(* Logix 5000 project; controller DispersionPlc vendor 1 type 14 code 108 rev 34.11; software revision 34.01; part 5 of 22 *)
(* tags used below, declared in another part *)
   catalyst_Target_Wgt_Lb_Min : REAL;
   D_Alarm_11_Timer : TIMER;
   D_Alarm_9_Timer : TIMER;
   D_AlarmTimers : TIMER[200];
   D_AlarmTimers2 : TIMER[100];
   DPT_4303_Warn : REAL;
   ONS : BOOL[32];
   ZS_4301_timer : TIMER;
   ZS_4302_timer : TIMER;
   _JISdebug : DINT;
   AFB : BOOL;
   AFI : BOOL;
   AMMONIUM_START_ATTEMP : BOOL;
   BL_4310_AUX : ALIAS FOR Local:1:I.Data[1].2;
   BL_4310_RUN : ALIAS FOR Local:1:O.Data[0].2;
   BLANK64 : Stp64;
   Cat_Destination_K400 : BOOL;
   Cat_Destination_K400_ONS : BOOL;
   Cat_Destination_K400_PB : BOOL;
   Cat_Destination_T4301 : BOOL;
   Cat_Destination_T4301_ONS : BOOL;
   Cat_Destination_T4301_PB : BOOL;
   Cat_Isolation_Valve_Timer : TIMER;
   Cat_Purge_Transfer_K400 : Seq64;
   Cat_Purge_Transfer_T430X : Seq64;
   Cat_Recirc_Transfer_K400 : Seq64;
   Cat_Recirc_Transfer_T430X : Seq64;
   Cat_Tank_Destination : DINT;
   cat_target_weight_bypass : BOOL;
   catalyst_MaxFeedRate : REAL;
   CATALYST_RESET : BOOL;
   CATFLOW : TIMER;
   CE_4301 : REAL;
   ce_4301_High : REAL;
   ce_4301_Low : REAL;
   DispAlarmResetBit : BOOL;
   DispersionAlarms : BOOL[256];
   DPT_4301 : REAL;
   dpt_4301_High : REAL;
   DPT_4302 : REAL;
   dpt_4302_High : REAL;
   DPT_4303 : REAL;
   DPT_4303_High : REAL;
   Drum_Transfer : BOOL;
   Enable_Shortstop_Automation : BOOL;
   Estop_Bulk : ALIAS FOR Local:1:I.Data[33].5;
   Estop_Disp : ALIAS FOR Local:3:I.Data.1;
   Estop_Inx : ALIAS FOR Local:3:I.Data.3;
   Estop_Mcc : ALIAS FOR Local:3:I.Data.2;
   FE_4303 : REAL;
   FE_4303_Low : REAL;
   FE_4304 : REAL;
   FE_4304_Low : REAL;
   FE_4305 : REAL;
   FE_4305_LOW : REAL;
   GLOBAL_RESET : BOOL;
   HMI_4303_Timer : REAL;
   HMI_4304_Timer : REAL;
   HMI_Cat_Isolation_Valve_Timer : REAL;
   HMI_V4304_PumpSpeedScaleIn : REAL;
   K4_High_Temp : BOOL;
   K4_Low_Temp : BOOL;
   LAH_S4352_1 : ALIAS FOR Local:1:I.Data[27].13;
   Linked_Timer : TIMER;
   LS_4301 : ALIAS FOR Local:2:I.Data.10;
   LS_4302 : ALIAS FOR Local:2:I.Data.11;
   LS_4302_High : BOOL;
   LS_T53_High : ALIAS FOR Local:1:I.Data[27].12;
   MCR_Bulk : ALIAS FOR Local:1:I.Data[33].4;
   MIXER_A_4301_RUN : ALIAS FOR Local:1:O.Data[0].0;
   MIXER_A_4303_AUX : ALIAS FOR Local:1:I.Data[1].4;
   MIXER_A_4303_RUN : ALIAS FOR Local:1:O.Data[0].4;
   MIXER_A_4304_AUX : ALIAS FOR Local:1:I.Data[1].16;
   MIXER_A_4304_RUN : ALIAS FOR Local:1:O.Data[0].16;
   MIXER_T_4301_AUX : ALIAS FOR Local:1:I.Data[1].0;
   MMI_Disp_Alarm_Reset_Pb : BOOL;
   MMI_Dispersion_Interlock_Bypass : BOOL;
   Mon_Tank_Destination : DINT;
   PS_AirMakeup : ALIAS FOR Local:1:I.Data[33].3;
   PUMP_P_4305_AUX : ALIAS FOR Local:1:I.Data[1].7;
   PUMP_P_4305_RUN : ALIAS FOR Local:1:O.Data[0].7;
   RG_T52 : REAL;
   RG_T52_Warn : REAL;
   RG_T53 : REAL;
   RG_T53_Warn : REAL;
   SPARE_I304 : ALIAS FOR Local:3:I.Data.4;
   SPARE_I305 : ALIAS FOR Local:3:I.Data.5;
   SPARE_O510 : ALIAS FOR Local:5:O.Data.10;
   SRT_PB_BL_4310 : ALIAS FOR Local:2:I.Data.13;
   ST_K400_1 : REAL;
   SV_4304 : ALIAS FOR Local:5:O.Data.11;
   SV_4304_02 : BOOL;
   SV_4304_02_Enable_PB : BOOL;
   SV_4304_03 : BOOL;
   SV_4304_03_Enable_PB : BOOL;
   T4301_Mixer : VFD;
   T4302_Mixer : VFD;
   T52_Mixer : VFD;
   Tank_Destination_ONS1 : BOOL;
   Task_Permissive : DINT[2];
   TE_4301A : ALIAS FOR Local:8:I.Ch0Data;
   Te_4301A_High : REAL;
   TE_4302A : ALIAS FOR Local:8:I.Ch5Data;
   TE_4302A_High : REAL;
   TE_4304 : ALIAS FOR Local:9:I.Ch5Data;
   TE_4304_High : REAL;
   TO_ALARM_MSG_DINT : DINT;
   TOGGLE : BOOL;
   Trans_Pump_P52_Aux : ALIAS FOR Local:1:I.Data[33].0;
   Trans_Pump_P53_Aux : ALIAS FOR Local:1:I.Data[33].1;
   TRANS_PUMP_P_4301_AUX : ALIAS FOR Local:1:I.Data[1].1;
   TRANS_PUMP_P_4301_RUN : ALIAS FOR Local:1:O.Data[0].1;
   TRANS_PUMP_P_4302_AUX : ALIAS FOR Local:1:I.Data[1].3;
   TRANS_PUMP_P_4302_RUN : ALIAS FOR Local:1:O.Data[0].3;
   Trans_Pump_T52_Run : ALIAS FOR Local:1:O.Data[13].1;
   Trans_Pump_T53_Run : ALIAS FOR Local:1:O.Data[13].2;
   V4304_Pump : VFD;
   W4303_Pump : VFD;
   XI_K400_1 : BOOL;
   XV_4301 : ALIAS FOR Local:5:O.Data.0;
   XV_4302 : ALIAS FOR Local:5:O.Data.1;
   XV_4303_01 : ALIAS FOR Local:5:O.Data.3;
   XV_4304 : ALIAS FOR Local:5:O.Data.4;
   XV_4304_02 : BOOL;
   XV_4304_03 : BOOL;
   XV_4304_04 : BOOL;
   XV_5201 : ALIAS FOR Local:1:O.Data[12].8;
   XV_5202 : ALIAS FOR Local:1:O.Data[12].9;
   XV_5301 : ALIAS FOR Local:1:O.Data[12].6;
   XV_5302 : ALIAS FOR Local:1:O.Data[12].7;
   XV_K400_04_SEQCLOSE : BOOL;
   XV_K400_04_SEQOPEN : BOOL;
   ZSC_4301 : ALIAS FOR Local:2:I.Data.1;
   ZSC_4302 : ALIAS FOR Local:2:I.Data.3;
   ZSC_4303_1 : ALIAS FOR Local:2:I.Data.7;
   ZSC_4304 : ALIAS FOR Local:2:I.Data.9;
   ZSC_4304_02 : BOOL;
   ZSC_4304_03 : BOOL;
   ZSC_5201 : ALIAS FOR Local:1:I.Data[27].5;
   ZSC_5202 : ALIAS FOR Local:1:I.Data[27].7;
   ZSC_5301 : ALIAS FOR Local:1:I.Data[27].9;
   ZSC_5302 : ALIAS FOR Local:1:I.Data[27].11;
   ZSC_K400_04 : BOOL;
   ZSO_4301 : ALIAS FOR Local:2:I.Data.0;
   ZSO_4302 : ALIAS FOR Local:2:I.Data.2;
   ZSO_4303_1 : ALIAS FOR Local:2:I.Data.6;
   ZSO_4304 : ALIAS FOR Local:2:I.Data.8;
   ZSO_4304_02 : BOOL;
   ZSO_4304_03 : BOOL;
   ZSO_4304_04 : BOOL;
   ZSO_5201 : ALIAS FOR Local:1:I.Data[27].4;
   ZSO_5202 : ALIAS FOR Local:1:I.Data[27].6;
   ZSO_5301 : ALIAS FOR Local:1:I.Data[27].8;
   ZSO_5302 : ALIAS FOR Local:1:I.Data[27].10;
   ZSO_K400_04 : BOOL;
(* MainProgram, continued *)

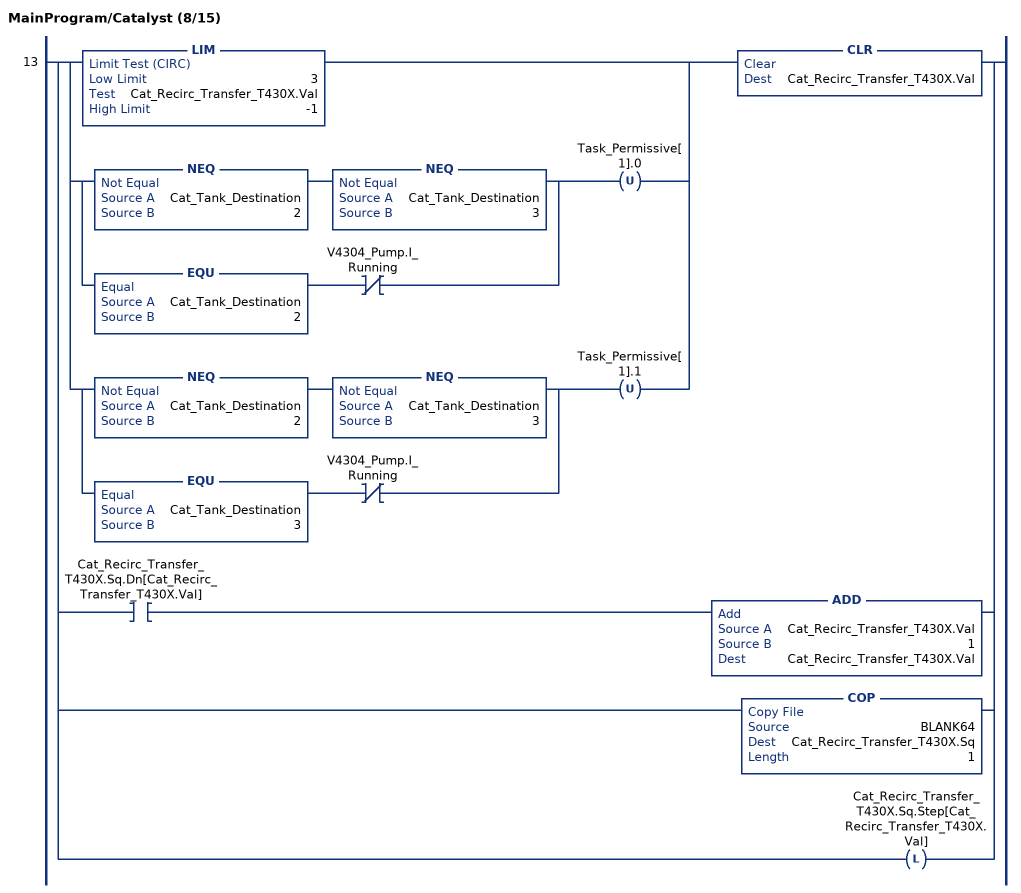
   [picture p69: MainProgram/Catalyst rungs 13-13]
   13: [[LIM(3,Cat_Recirc_Transfer_T430X.Val,-1) ,[NEQ(Cat_Tank_Destination,2) NEQ(Cat_Tank_Destination,3) ,EQU(Cat_Tank_Destination,2) XIO(V4304_Pump.I_Running) ] OTU(Task_Permissive[1].0) ,[NEQ(Cat_Tank_Destination,2) NEQ(Cat_Tank_Destination,3) ,EQU(Cat_Tank_Destination,3) XIO(V4304_Pump.I_Running) ] OTU(Task_Permissive[1].1) ] CLR(Cat_Recirc_Transfer_T430X.Val) ,XIC(Cat_Recirc_Transfer_T430X.Sq.Dn[Cat_Recirc_Transfer_T430X.Val]) ADD(Cat_Recirc_Transfer_T430X.Val,1,Cat_Recirc_Transfer_T430X.Val) ,COP(BLANK64,Cat_Recirc_Transfer_T430X.Sq,1) ,OTL(Cat_Recirc_Transfer_T430X.Sq.Step[Cat_Recirc_Transfer_T430X.Val]) ];
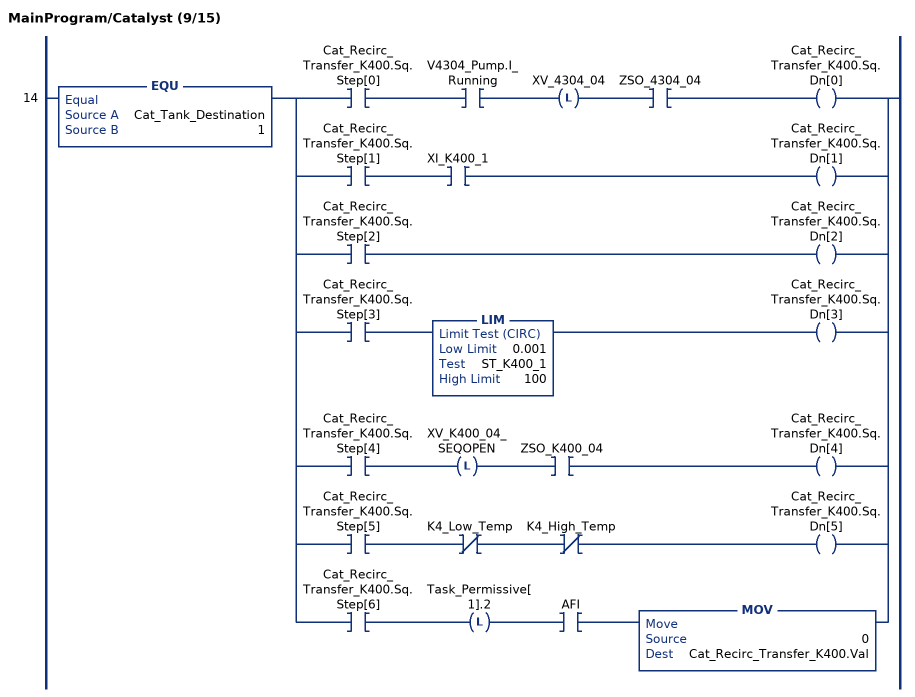
   14: EQU(Cat_Tank_Destination,1)[XIC(Cat_Recirc_Transfer_K400.Sq.Step[0]) XIC(V4304_Pump.I_Running) OTL(XV_4304_04) XIC(ZSO_4304_04) OTE(Cat_Recirc_Transfer_K400.Sq.Dn[0]) ,XIC(Cat_Recirc_Transfer_K400.Sq.Step[1]) XIC(XI_K400_1) OTE(Cat_Recirc_Transfer_K400.Sq.Dn[1]) ,XIC(Cat_Recirc_Transfer_K400.Sq.Step[2]) OTE(Cat_Recirc_Transfer_K400.Sq.Dn[2]) ,XIC(Cat_Recirc_Transfer_K400.Sq.Step[3]) LIM(0.001,ST_K400_1,100) OTE(Cat_Recirc_Transfer_K400.Sq.Dn[3]) ,XIC(Cat_Recirc_Transfer_K400.Sq.Step[4]) OTL(XV_K400_04_SEQOPEN) XIC(ZSO_K400_04) OTE(Cat_Recirc_Transfer_K400.Sq.Dn[4]) ,XIC(Cat_Recirc_Transfer_K400.Sq.Step[5]) XIO(K4_Low_Temp) XIO(K4_High_Temp) OTE(Cat_Recirc_Transfer_K400.Sq.Dn[5]) ,XIC(Cat_Recirc_Transfer_K400.Sq.Step[6]) OTL(Task_Permissive[1].2) XIC(AFI) MOV(0,Cat_Recirc_Transfer_K400.Val) ];
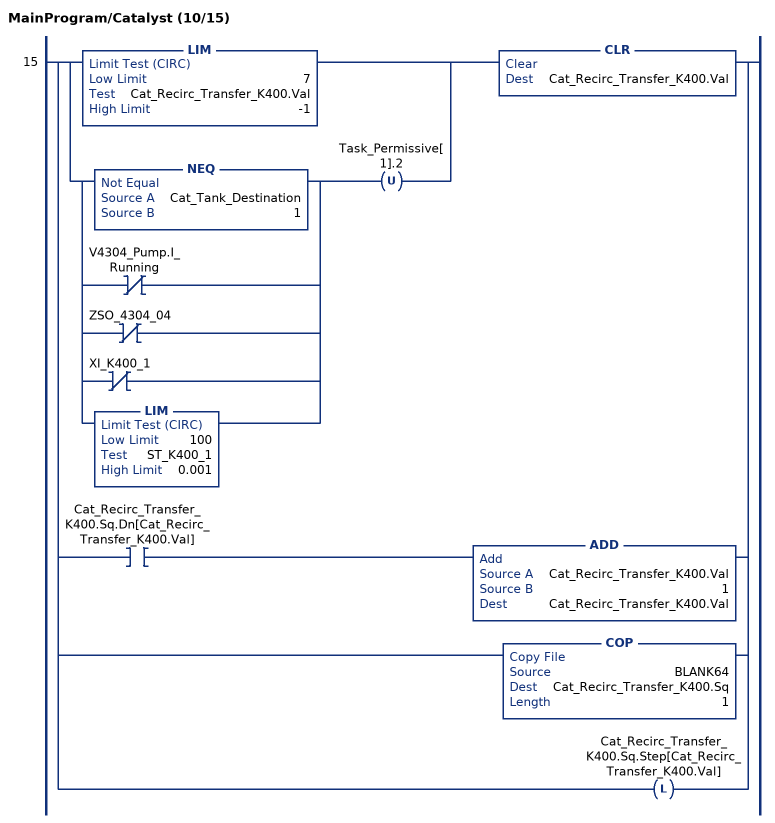
   15: [[LIM(7,Cat_Recirc_Transfer_K400.Val,-1) ,[NEQ(Cat_Tank_Destination,1) ,XIO(V4304_Pump.I_Running) ,XIO(ZSO_4304_04) ,XIO(XI_K400_1) ,LIM(100,ST_K400_1,0.001) ] OTU(Task_Permissive[1].2) ] CLR(Cat_Recirc_Transfer_K400.Val) ,XIC(Cat_Recirc_Transfer_K400.Sq.Dn[Cat_Recirc_Transfer_K400.Val]) ADD(Cat_Recirc_Transfer_K400.Val,1,Cat_Recirc_Transfer_K400.Val) ,COP(BLANK64,Cat_Recirc_Transfer_K400.Sq,1) ,OTL(Cat_Recirc_Transfer_K400.Sq.Step[Cat_Recirc_Transfer_K400.Val]) ];
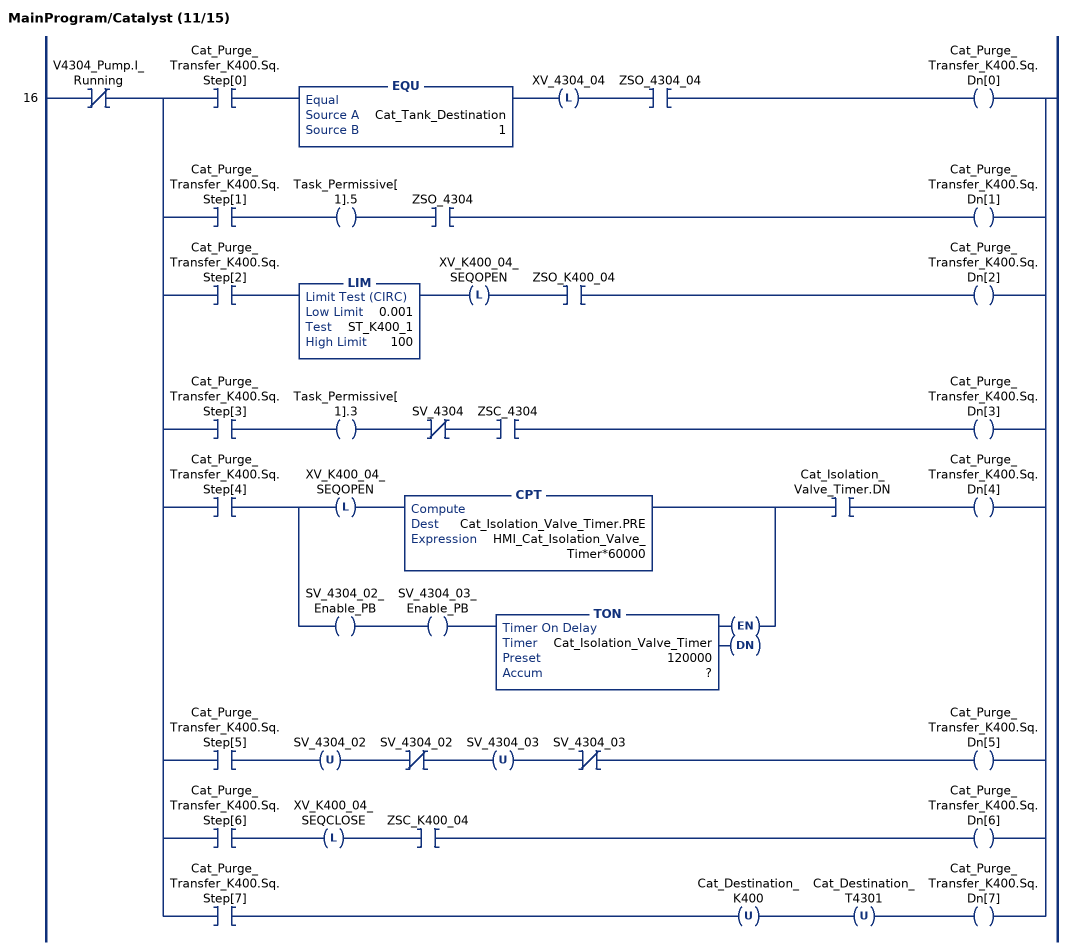
   16: XIO(V4304_Pump.I_Running)[XIC(Cat_Purge_Transfer_K400.Sq.Step[0]) EQU(Cat_Tank_Destination,1) OTL(XV_4304_04) XIC(ZSO_4304_04) OTE(Cat_Purge_Transfer_K400.Sq.Dn[0]) ,XIC(Cat_Purge_Transfer_K400.Sq.Step[1]) OTE(Task_Permissive[1].5) XIC(ZSO_4304) OTE(Cat_Purge_Transfer_K400.Sq.Dn[1]) ,XIC(Cat_Purge_Transfer_K400.Sq.Step[2]) LIM(0.001,ST_K400_1,100) OTL(XV_K400_04_SEQOPEN) XIC(ZSO_K400_04) OTE(Cat_Purge_Transfer_K400.Sq.Dn[2]) ,XIC(Cat_Purge_Transfer_K400.Sq.Step[3]) OTE(Task_Permissive[1].3) XIO(SV_4304) XIC(ZSC_4304) OTE(Cat_Purge_Transfer_K400.Sq.Dn[3]) ,XIC(Cat_Purge_Transfer_K400.Sq.Step[4]) [OTL(XV_K400_04_SEQOPEN) CPT(Cat_Isolation_Valve_Timer.PRE,HMI_Cat_Isolation_Valve_Timer*60000) ,OTE(SV_4304_02_Enable_PB) OTE(SV_4304_03_Enable_PB) TON(Cat_Isolation_Valve_Timer,?,?) ] XIC(Cat_Isolation_Valve_Timer.DN) OTE(Cat_Purge_Transfer_K400.Sq.Dn[4]) ,XIC(Cat_Purge_Transfer_K400.Sq.Step[5]) OTU(SV_4304_02) XIO(SV_4304_02) OTU(SV_4304_03) XIO(SV_4304_03) OTE(Cat_Purge_Transfer_K400.Sq.Dn[5]) ,XIC(Cat_Purge_Transfer_K400.Sq.Step[6]) OTL(XV_K400_04_SEQCLOSE) XIC(ZSC_K400_04) OTE(Cat_Purge_Transfer_K400.Sq.Dn[6]) ,XIC(Cat_Purge_Transfer_K400.Sq.Step[7]) OTU(Cat_Destination_K400) OTU(Cat_Destination_T4301) OTE(Cat_Purge_Transfer_K400.Sq.Dn[7]) ];
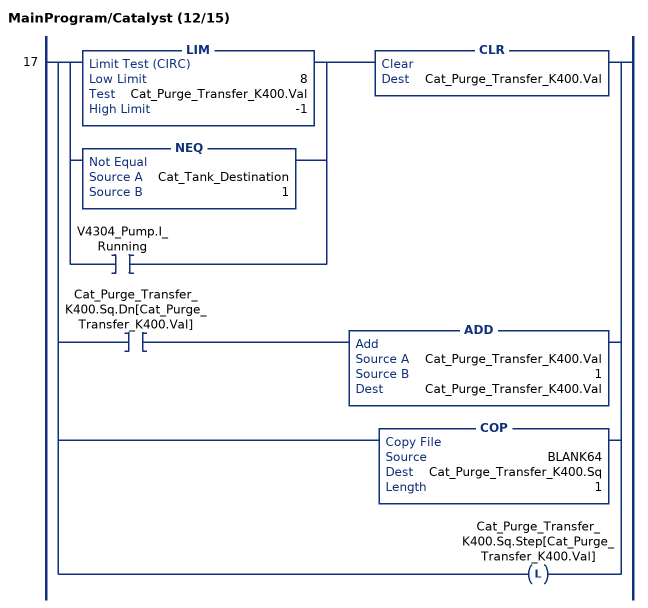
   17: [[LIM(8,Cat_Purge_Transfer_K400.Val,-1) ,NEQ(Cat_Tank_Destination,1) ,XIC(V4304_Pump.I_Running) ] CLR(Cat_Purge_Transfer_K400.Val) ,XIC(Cat_Purge_Transfer_K400.Sq.Dn[Cat_Purge_Transfer_K400.Val]) ADD(Cat_Purge_Transfer_K400.Val,1,Cat_Purge_Transfer_K400.Val) ,COP(BLANK64,Cat_Purge_Transfer_K400.Sq,1) ,OTL(Cat_Purge_Transfer_K400.Sq.Step[Cat_Purge_Transfer_K400.Val]) ];
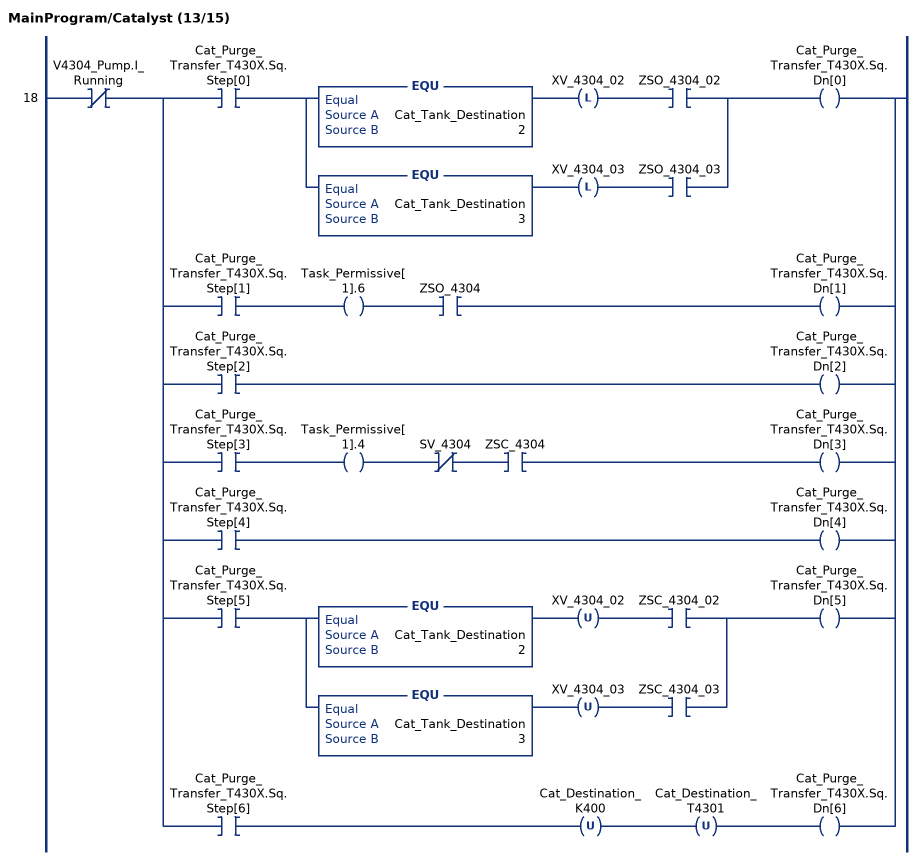
   18: XIO(V4304_Pump.I_Running)[XIC(Cat_Purge_Transfer_T430X.Sq.Step[0]) [EQU(Cat_Tank_Destination,2) OTL(XV_4304_02) XIC(ZSO_4304_02) ,EQU(Cat_Tank_Destination,3) OTL(XV_4304_03) XIC(ZSO_4304_03) ] OTE(Cat_Purge_Transfer_T430X.Sq.Dn[0]) ,XIC(Cat_Purge_Transfer_T430X.Sq.Step[1]) OTE(Task_Permissive[1].6) XIC(ZSO_4304) OTE(Cat_Purge_Transfer_T430X.Sq.Dn[1]) ,XIC(Cat_Purge_Transfer_T430X.Sq.Step[2]) OTE(Cat_Purge_Transfer_T430X.Sq.Dn[2]) ,XIC(Cat_Purge_Transfer_T430X.Sq.Step[3]) OTE(Task_Permissive[1].4) XIO(SV_4304) XIC(ZSC_4304) OTE(Cat_Purge_Transfer_T430X.Sq.Dn[3]) ,XIC(Cat_Purge_Transfer_T430X.Sq.Step[4]) OTE(Cat_Purge_Transfer_T430X.Sq.Dn[4]) ,XIC(Cat_Purge_Transfer_T430X.Sq.Step[5]) [EQU(Cat_Tank_Destination,2) OTU(XV_4304_02) XIC(ZSC_4304_02) ,EQU(Cat_Tank_Destination,3) OTU(XV_4304_03) XIC(ZSC_4304_03) ] OTE(Cat_Purge_Transfer_T430X.Sq.Dn[5]) ,XIC(Cat_Purge_Transfer_T430X.Sq.Step[6]) OTU(Cat_Destination_K400) OTU(Cat_Destination_T4301) OTE(Cat_Purge_Transfer_T430X.Sq.Dn[6]) ];
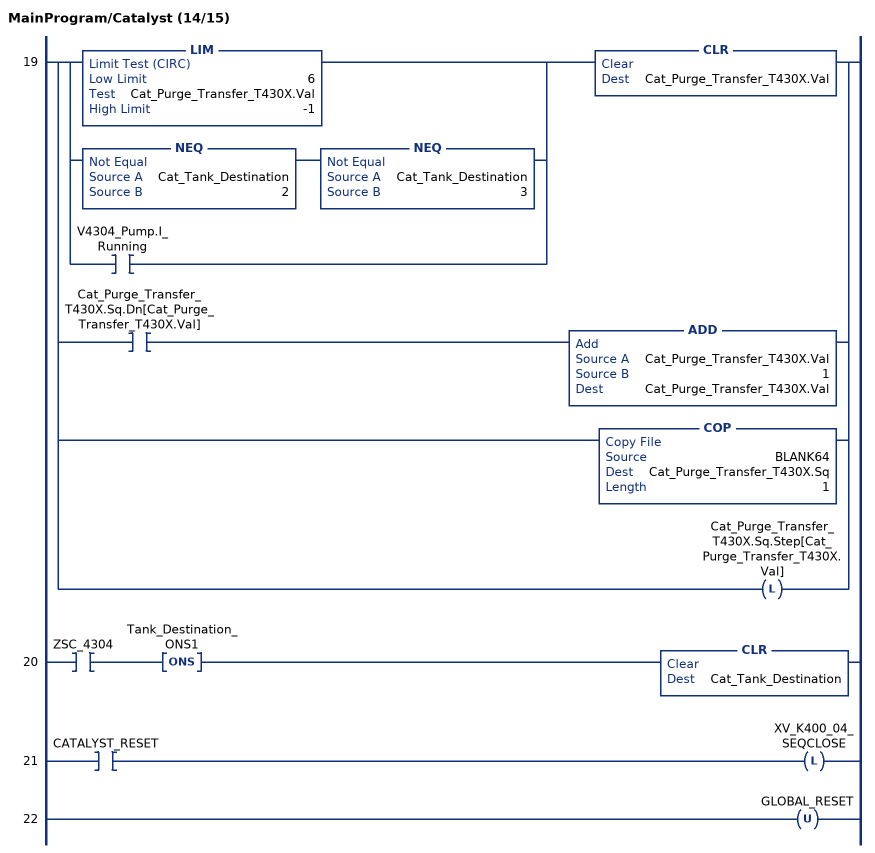
   19: [[LIM(6,Cat_Purge_Transfer_T430X.Val,-1) ,NEQ(Cat_Tank_Destination,2) NEQ(Cat_Tank_Destination,3) ,XIC(V4304_Pump.I_Running) ] CLR(Cat_Purge_Transfer_T430X.Val) ,XIC(Cat_Purge_Transfer_T430X.Sq.Dn[Cat_Purge_Transfer_T430X.Val]) ADD(Cat_Purge_Transfer_T430X.Val,1,Cat_Purge_Transfer_T430X.Val) ,COP(BLANK64,Cat_Purge_Transfer_T430X.Sq,1) ,OTL(Cat_Purge_Transfer_T430X.Sq.Step[Cat_Purge_Transfer_T430X.Val]) ];
   20: XIC(ZSC_4304)ONS(Tank_Destination_ONS1)CLR(Cat_Tank_Destination);
   21: XIC(CATALYST_RESET)OTL(XV_K400_04_SEQCLOSE);
   22: OTU(GLOBAL_RESET);
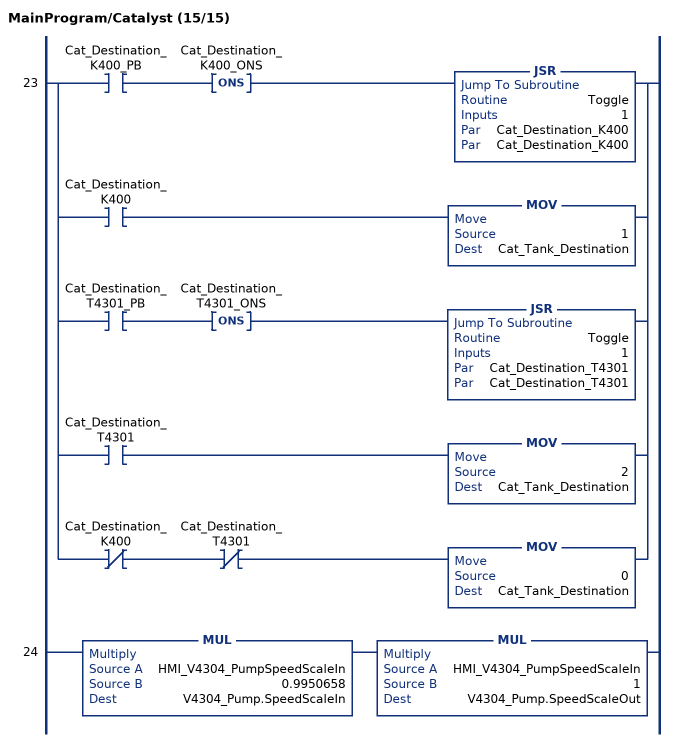
   23: [[XIC(Cat_Destination_K400_PB) ONS(Cat_Destination_K400_ONS) JSR(Toggle,1,Cat_Destination_K400,Cat_Destination_K400) ,XIC(Cat_Destination_K400) MOV(1,Cat_Tank_Destination) ] ,[XIC(Cat_Destination_T4301_PB) ONS(Cat_Destination_T4301_ONS) JSR(Toggle,1,Cat_Destination_T4301,Cat_Destination_T4301) ,XIC(Cat_Destination_T4301) MOV(2,Cat_Tank_Destination) ] ,XIO(Cat_Destination_K400) XIO(Cat_Destination_T4301) MOV(0,Cat_Tank_Destination) ];
   24: MUL(HMI_V4304_PumpSpeedScaleIn,0.9950658,V4304_Pump.SpeedScaleIn)MUL(HMI_V4304_PumpSpeedScaleIn,1,V4304_Pump.SpeedScaleOut);
END_ROUTINE

ROUTINE Dispersion_Alarms   (* ladder *)
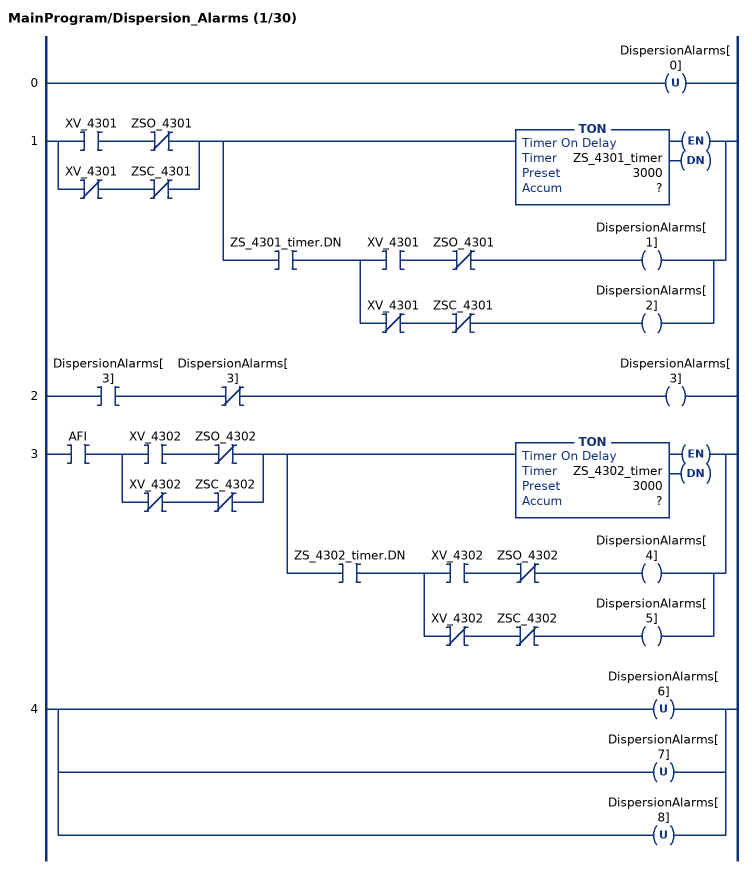
   0: OTU(DispersionAlarms[0]);
   1: [XIC(XV_4301) XIO(ZSO_4301) ,XIO(XV_4301) XIO(ZSC_4301) ][TON(ZS_4301_timer,?,?) ,XIC(ZS_4301_timer.DN) [XIC(XV_4301) XIO(ZSO_4301) OTE(DispersionAlarms[1]) ,XIO(XV_4301) XIO(ZSC_4301) OTE(DispersionAlarms[2]) ] ];
   2: XIC(DispersionAlarms[3])XIO(DispersionAlarms[3])OTE(DispersionAlarms[3]);
   3: XIC(AFI)[XIC(XV_4302) XIO(ZSO_4302) ,XIO(XV_4302) XIO(ZSC_4302) ][TON(ZS_4302_timer,?,?) ,XIC(ZS_4302_timer.DN) [XIC(XV_4302) XIO(ZSO_4302) OTE(DispersionAlarms[4]) ,XIO(XV_4302) XIO(ZSC_4302) OTE(DispersionAlarms[5]) ] ];
   4: [OTU(DispersionAlarms[6]) ,OTU(DispersionAlarms[7]) ,OTU(DispersionAlarms[8]) ];
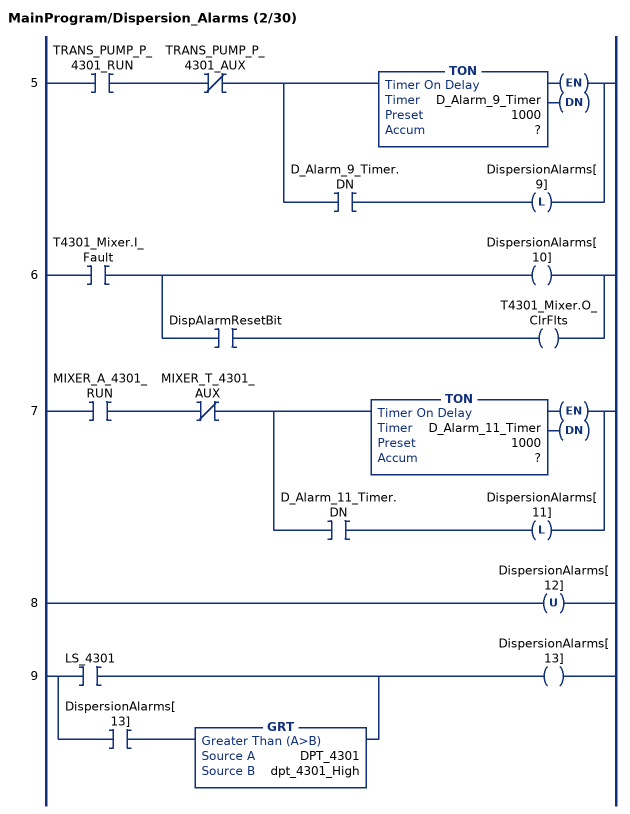
   5: XIC(TRANS_PUMP_P_4301_RUN)XIO(TRANS_PUMP_P_4301_AUX)[TON(D_Alarm_9_Timer,?,?) ,XIC(D_Alarm_9_Timer.DN) OTL(DispersionAlarms[9]) ];
   6: XIC(T4301_Mixer.I_Fault)[OTE(DispersionAlarms[10]) ,XIC(DispAlarmResetBit) OTE(T4301_Mixer.O_ClrFlts) ];
   7: XIC(MIXER_A_4301_RUN)XIO(MIXER_T_4301_AUX)[TON(D_Alarm_11_Timer,?,?) ,XIC(D_Alarm_11_Timer.DN) OTL(DispersionAlarms[11]) ];
   8: OTU(DispersionAlarms[12]);
   9: [XIC(LS_4301) ,XIC(DispersionAlarms[13]) GRT(DPT_4301,dpt_4301_High) ]OTE(DispersionAlarms[13]);
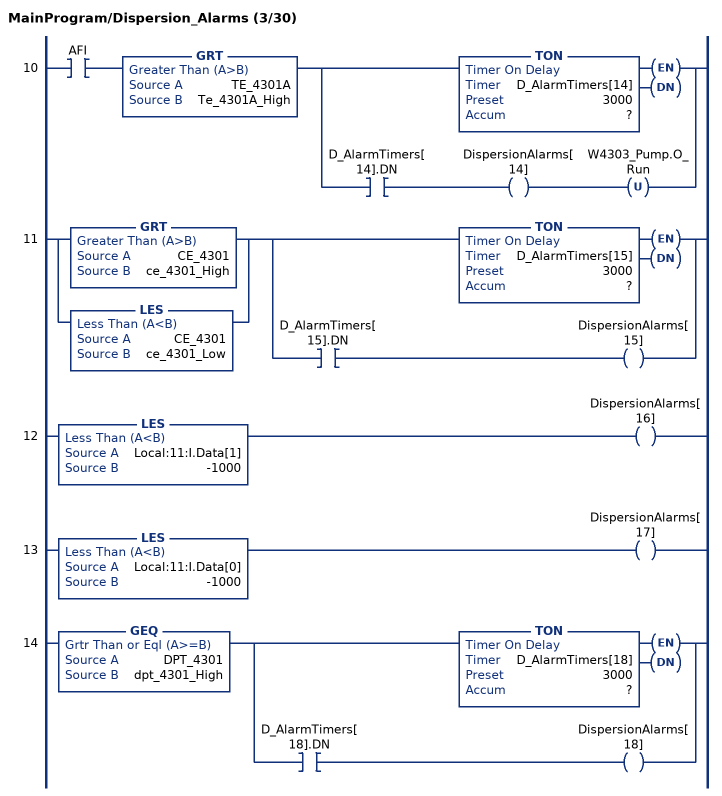
   10: XIC(AFI)GRT(TE_4301A,Te_4301A_High)[TON(D_AlarmTimers[14],?,?) ,XIC(D_AlarmTimers[14].DN) OTE(DispersionAlarms[14]) OTU(W4303_Pump.O_Run) ];
   11: [GRT(CE_4301,ce_4301_High) ,LES(CE_4301,ce_4301_Low) ][TON(D_AlarmTimers[15],?,?) ,XIC(D_AlarmTimers[15].DN) OTE(DispersionAlarms[15]) ];
   12: LES(Local:11:I.Data[1],-1000)OTE(DispersionAlarms[16]);
   13: LES(Local:11:I.Data[0],-1000)OTE(DispersionAlarms[17]);
   14: GEQ(DPT_4301,dpt_4301_High)[TON(D_AlarmTimers[18],?,?) ,XIC(D_AlarmTimers[18].DN) OTE(DispersionAlarms[18]) ];
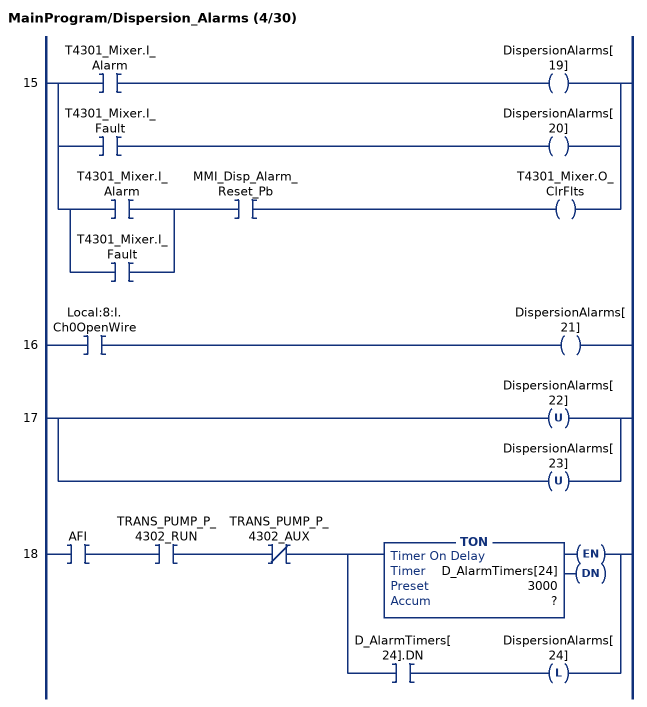
   15: [XIC(T4301_Mixer.I_Alarm) OTE(DispersionAlarms[19]) ,XIC(T4301_Mixer.I_Fault) OTE(DispersionAlarms[20]) ,[XIC(T4301_Mixer.I_Alarm) ,XIC(T4301_Mixer.I_Fault) ] XIC(MMI_Disp_Alarm_Reset_Pb) OTE(T4301_Mixer.O_ClrFlts) ];
   16: XIC(Local:8:I.Ch0OpenWire)OTE(DispersionAlarms[21]);
   17: [OTU(DispersionAlarms[22]) ,OTU(DispersionAlarms[23]) ];
   18: XIC(AFI)XIC(TRANS_PUMP_P_4302_RUN)XIO(TRANS_PUMP_P_4302_AUX)[TON(D_AlarmTimers[24],?,?) ,XIC(D_AlarmTimers[24].DN) OTL(DispersionAlarms[24]) ];
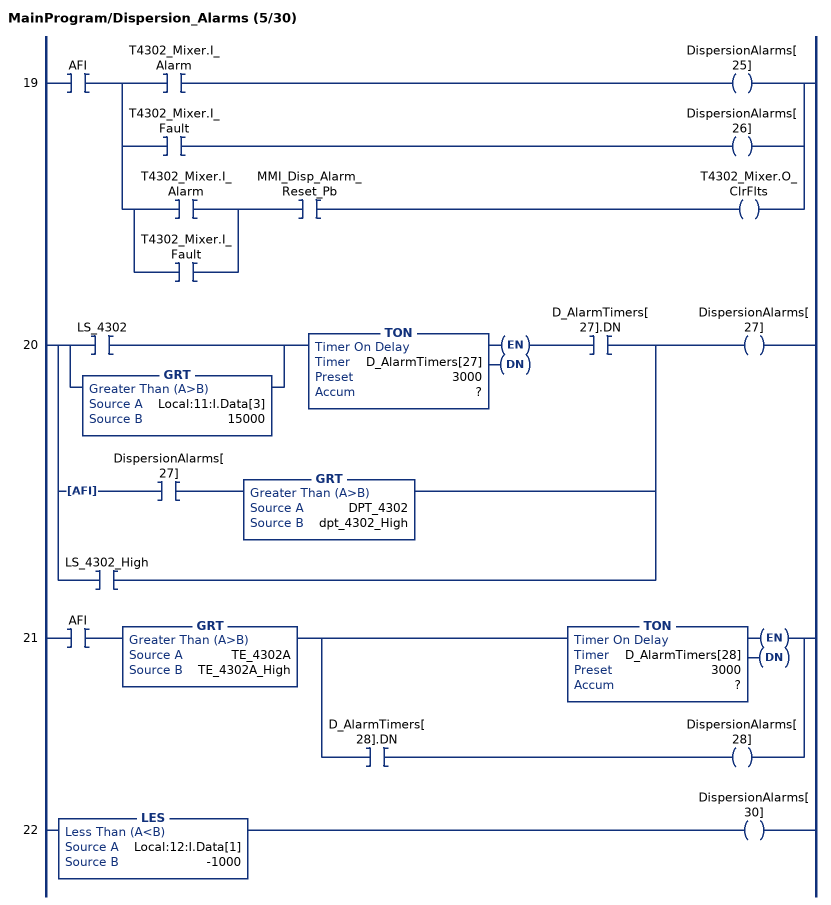
   19: XIC(AFI)[XIC(T4302_Mixer.I_Alarm) OTE(DispersionAlarms[25]) ,XIC(T4302_Mixer.I_Fault) OTE(DispersionAlarms[26]) ,[XIC(T4302_Mixer.I_Alarm) ,XIC(T4302_Mixer.I_Fault) ] XIC(MMI_Disp_Alarm_Reset_Pb) OTE(T4302_Mixer.O_ClrFlts) ];
   20: [[XIC(LS_4302) ,GRT(Local:11:I.Data[3],15000) ] TON(D_AlarmTimers[27],?,?) XIC(D_AlarmTimers[27].DN) ,AFI() XIC(DispersionAlarms[27]) GRT(DPT_4302,dpt_4302_High) ,XIC(LS_4302_High) ]OTE(DispersionAlarms[27]);
   21: XIC(AFI)GRT(TE_4302A,TE_4302A_High)[TON(D_AlarmTimers[28],?,?) ,XIC(D_AlarmTimers[28].DN) OTE(DispersionAlarms[28]) ];
   22: LES(Local:12:I.Data[1],-1000)OTE(DispersionAlarms[30]);
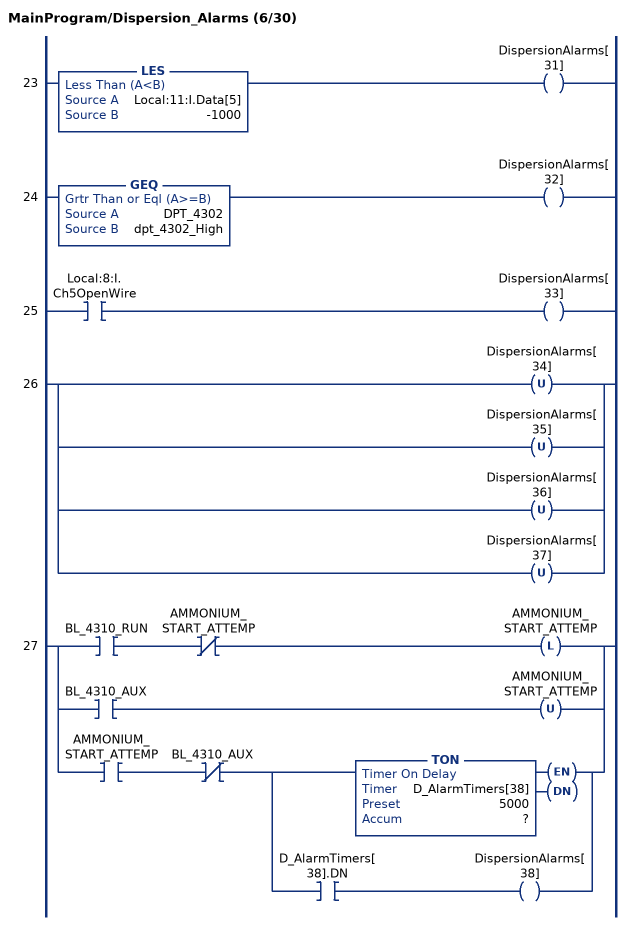
   23: LES(Local:11:I.Data[5],-1000)OTE(DispersionAlarms[31]);
   24: GEQ(DPT_4302,dpt_4302_High)OTE(DispersionAlarms[32]);
   25: XIC(Local:8:I.Ch5OpenWire)OTE(DispersionAlarms[33]);
   26: [OTU(DispersionAlarms[34]) ,OTU(DispersionAlarms[35]) ,OTU(DispersionAlarms[36]) ,OTU(DispersionAlarms[37]) ];
   27: [XIC(BL_4310_RUN) XIO(AMMONIUM_START_ATTEMP) OTL(AMMONIUM_START_ATTEMP) ,XIC(BL_4310_AUX) OTU(AMMONIUM_START_ATTEMP) ,XIC(AMMONIUM_START_ATTEMP) XIO(BL_4310_AUX) [TON(D_AlarmTimers[38],?,?) ,XIC(D_AlarmTimers[38].DN) OTE(DispersionAlarms[38]) ] ];
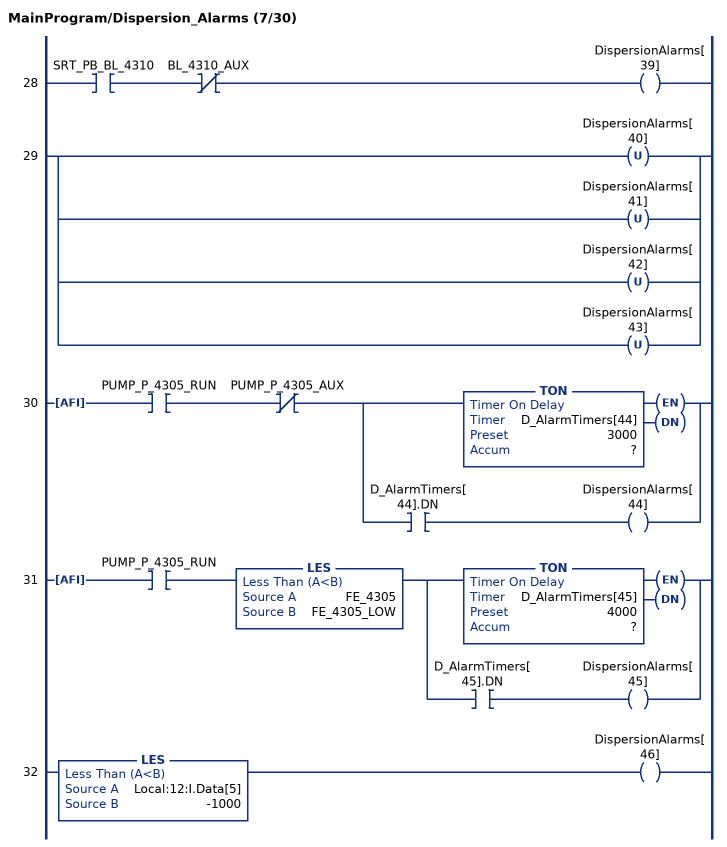
   28: XIC(SRT_PB_BL_4310)XIO(BL_4310_AUX)OTE(DispersionAlarms[39]);
   29: [OTU(DispersionAlarms[40]) ,OTU(DispersionAlarms[41]) ,OTU(DispersionAlarms[42]) ,OTU(DispersionAlarms[43]) ];
   30: AFI()XIC(PUMP_P_4305_RUN)XIO(PUMP_P_4305_AUX)[TON(D_AlarmTimers[44],?,?) ,XIC(D_AlarmTimers[44].DN) OTE(DispersionAlarms[44]) ];
   31: AFI()XIC(PUMP_P_4305_RUN)LES(FE_4305,FE_4305_LOW)[TON(D_AlarmTimers[45],?,?) ,XIC(D_AlarmTimers[45].DN) OTE(DispersionAlarms[45]) ];
   32: LES(Local:12:I.Data[5],-1000)OTE(DispersionAlarms[46]);
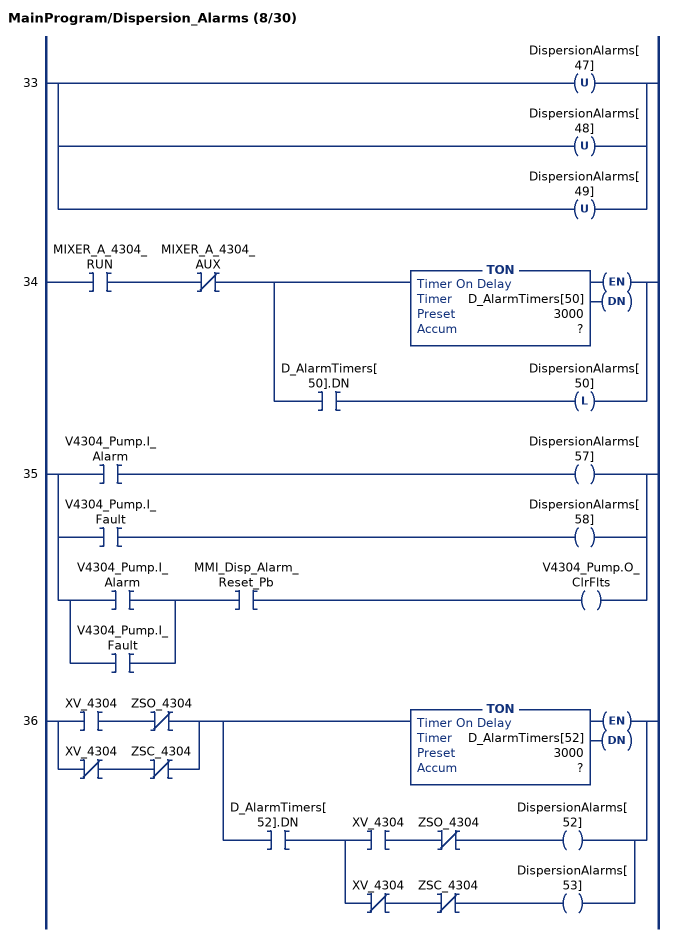
   33: [OTU(DispersionAlarms[47]) ,OTU(DispersionAlarms[48]) ,OTU(DispersionAlarms[49]) ];
   34: XIC(MIXER_A_4304_RUN)XIO(MIXER_A_4304_AUX)[TON(D_AlarmTimers[50],?,?) ,XIC(D_AlarmTimers[50].DN) OTL(DispersionAlarms[50]) ];
   35: [XIC(V4304_Pump.I_Alarm) OTE(DispersionAlarms[57]) ,XIC(V4304_Pump.I_Fault) OTE(DispersionAlarms[58]) ,[XIC(V4304_Pump.I_Alarm) ,XIC(V4304_Pump.I_Fault) ] XIC(MMI_Disp_Alarm_Reset_Pb) OTE(V4304_Pump.O_ClrFlts) ];
   36: [XIC(XV_4304) XIO(ZSO_4304) ,XIO(XV_4304) XIO(ZSC_4304) ][TON(D_AlarmTimers[52],?,?) ,XIC(D_AlarmTimers[52].DN) [XIC(XV_4304) XIO(ZSO_4304) OTE(DispersionAlarms[52]) ,XIO(XV_4304) XIO(ZSC_4304) OTE(DispersionAlarms[53]) ] ];
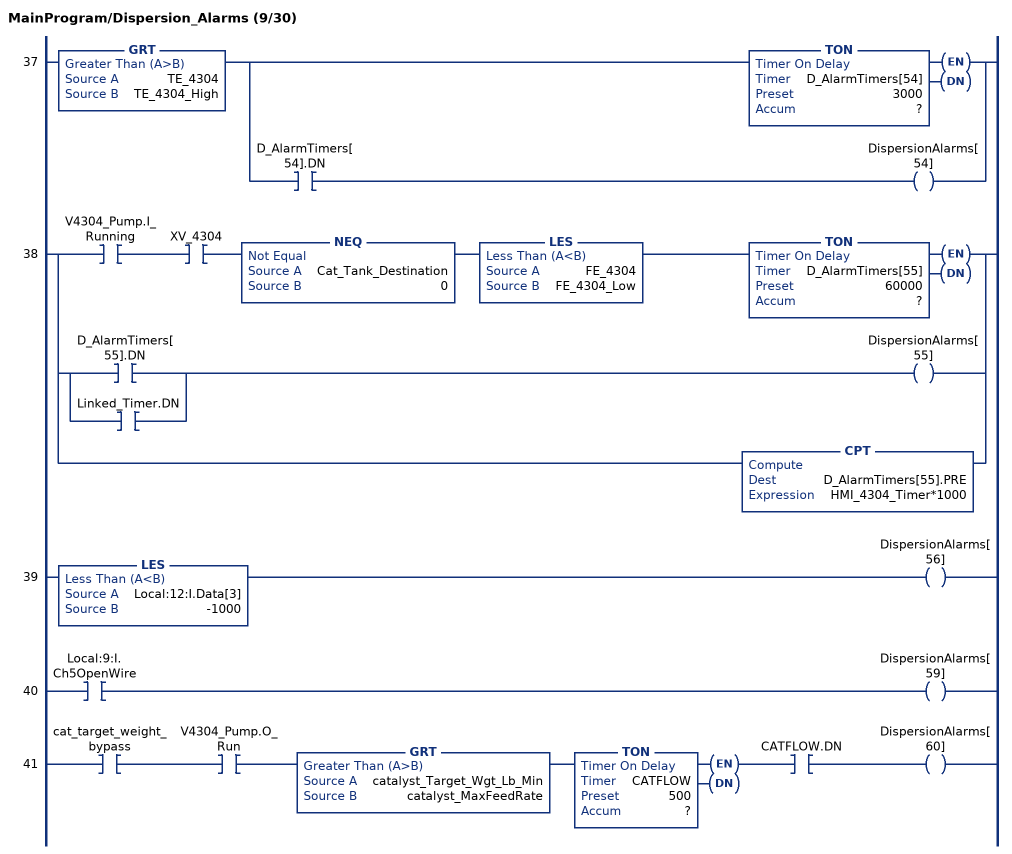
   37: GRT(TE_4304,TE_4304_High)[TON(D_AlarmTimers[54],?,?) ,XIC(D_AlarmTimers[54].DN) OTE(DispersionAlarms[54]) ];
   38: [XIC(V4304_Pump.I_Running) XIC(XV_4304) NEQ(Cat_Tank_Destination,0) LES(FE_4304,FE_4304_Low) TON(D_AlarmTimers[55],?,?) ,[XIC(D_AlarmTimers[55].DN) ,XIC(Linked_Timer.DN) ] OTE(DispersionAlarms[55]) ,CPT(D_AlarmTimers[55].PRE,HMI_4304_Timer*1000) ];
   39: LES(Local:12:I.Data[3],-1000)OTE(DispersionAlarms[56]);
   40: XIC(Local:9:I.Ch5OpenWire)OTE(DispersionAlarms[59]);
   41: XIC(cat_target_weight_bypass)XIC(V4304_Pump.O_Run)GRT(catalyst_Target_Wgt_Lb_Min,catalyst_MaxFeedRate)TON(CATFLOW,?,?)XIC(CATFLOW.DN)OTE(DispersionAlarms[60]);
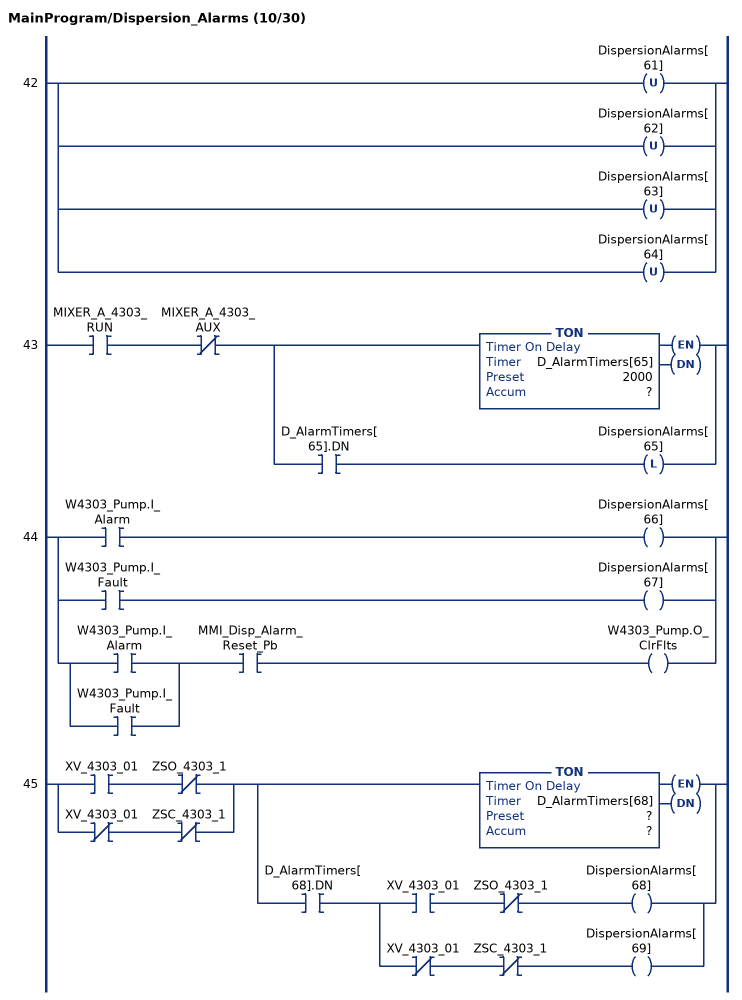
   42: [OTU(DispersionAlarms[61]) ,OTU(DispersionAlarms[62]) ,OTU(DispersionAlarms[63]) ,OTU(DispersionAlarms[64]) ];
   43: XIC(MIXER_A_4303_RUN)XIO(MIXER_A_4303_AUX)[TON(D_AlarmTimers[65],?,?) ,XIC(D_AlarmTimers[65].DN) OTL(DispersionAlarms[65]) ];
   44: [XIC(W4303_Pump.I_Alarm) OTE(DispersionAlarms[66]) ,XIC(W4303_Pump.I_Fault) OTE(DispersionAlarms[67]) ,[XIC(W4303_Pump.I_Alarm) ,XIC(W4303_Pump.I_Fault) ] XIC(MMI_Disp_Alarm_Reset_Pb) OTE(W4303_Pump.O_ClrFlts) ];
   45: [XIC(XV_4303_01) XIO(ZSO_4303_1) ,XIO(XV_4303_01) XIO(ZSC_4303_1) ][TON(D_AlarmTimers[68],?,?) ,XIC(D_AlarmTimers[68].DN) [XIC(XV_4303_01) XIO(ZSO_4303_1) OTE(DispersionAlarms[68]) ,XIO(XV_4303_01) XIO(ZSC_4303_1) OTE(DispersionAlarms[69]) ] ];
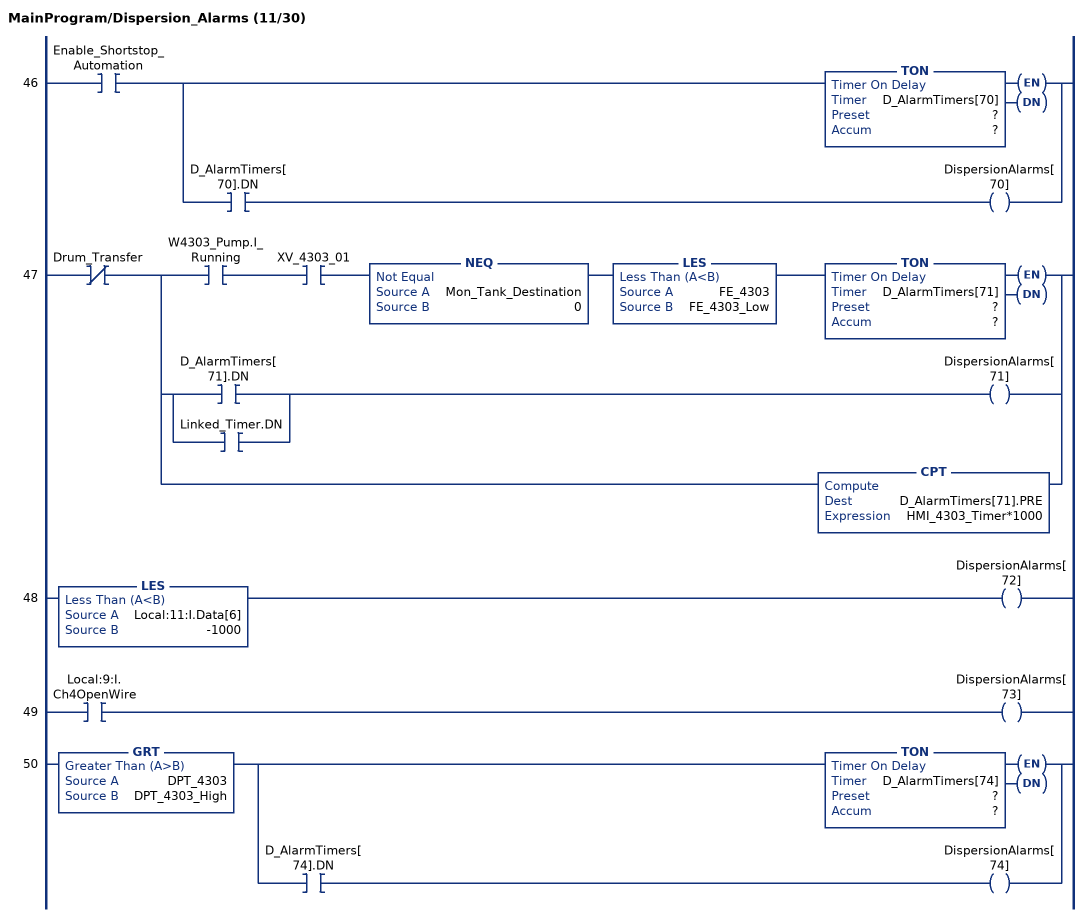
   46: XIC(Enable_Shortstop_Automation)[TON(D_AlarmTimers[70],?,?) ,XIC(D_AlarmTimers[70].DN) OTE(DispersionAlarms[70]) ];
   47: XIO(Drum_Transfer)[XIC(W4303_Pump.I_Running) XIC(XV_4303_01) NEQ(Mon_Tank_Destination,0) LES(FE_4303,FE_4303_Low) TON(D_AlarmTimers[71],?,?) ,[XIC(D_AlarmTimers[71].DN) ,XIC(Linked_Timer.DN) ] OTE(DispersionAlarms[71]) ,CPT(D_AlarmTimers[71].PRE,HMI_4303_Timer*1000) ];
   48: LES(Local:11:I.Data[6],-1000)OTE(DispersionAlarms[72]);
   49: XIC(Local:9:I.Ch4OpenWire)OTE(DispersionAlarms[73]);
   50: GRT(DPT_4303,DPT_4303_High)[TON(D_AlarmTimers[74],?,?) ,XIC(D_AlarmTimers[74].DN) OTE(DispersionAlarms[74]) ];
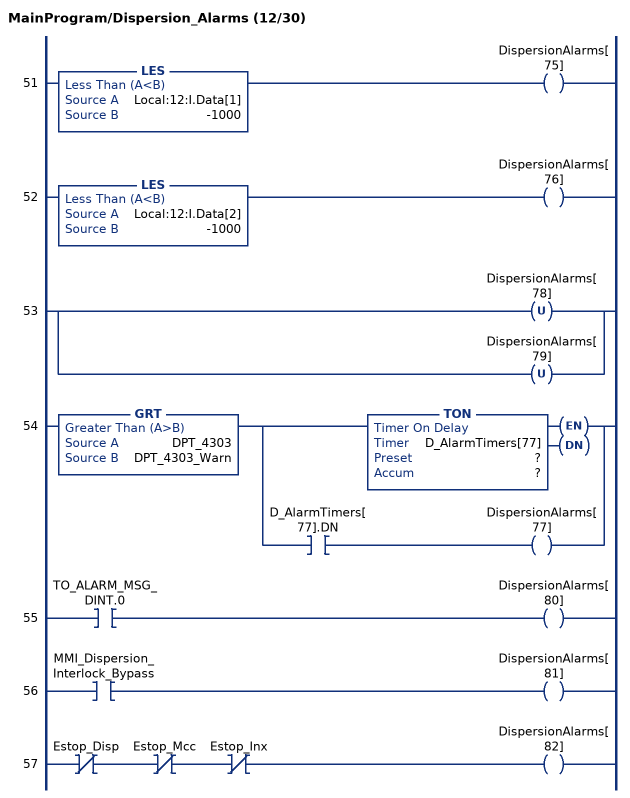
   51: LES(Local:12:I.Data[1],-1000)OTE(DispersionAlarms[75]);
   52: LES(Local:12:I.Data[2],-1000)OTE(DispersionAlarms[76]);
   53: [OTU(DispersionAlarms[78]) ,OTU(DispersionAlarms[79]) ];
   54: GRT(DPT_4303,DPT_4303_Warn)[TON(D_AlarmTimers[77],?,?) ,XIC(D_AlarmTimers[77].DN) OTE(DispersionAlarms[77]) ];
   55: XIC(TO_ALARM_MSG_DINT.0)OTE(DispersionAlarms[80]);
   56: XIC(MMI_Dispersion_Interlock_Bypass)OTE(DispersionAlarms[81]);
   57: XIO(Estop_Disp)XIO(Estop_Mcc)XIO(Estop_Inx)OTE(DispersionAlarms[82]);
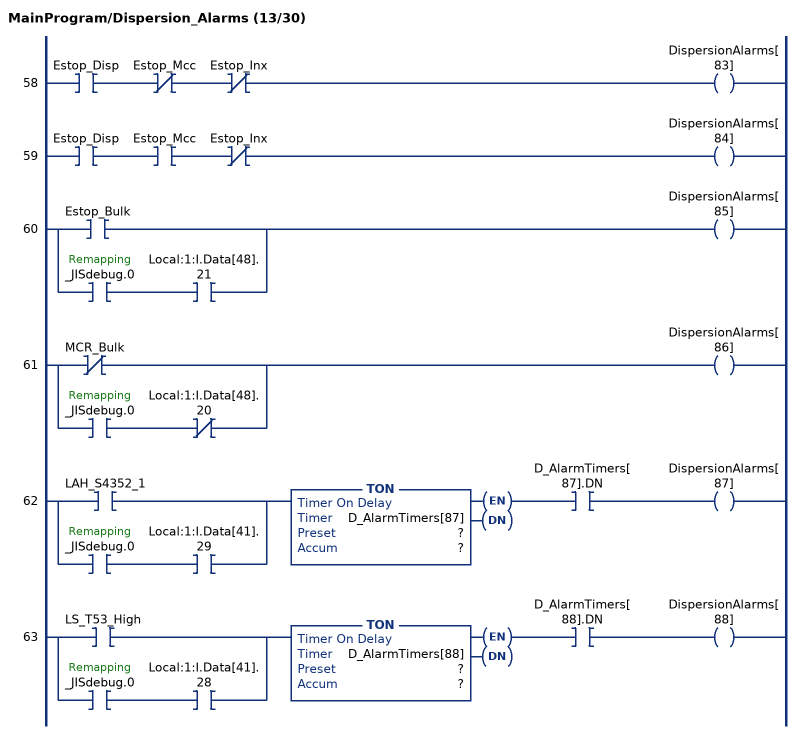
   58: XIC(Estop_Disp)XIO(Estop_Mcc)XIO(Estop_Inx)OTE(DispersionAlarms[83]);
   59: XIC(Estop_Disp)XIC(Estop_Mcc)XIO(Estop_Inx)OTE(DispersionAlarms[84]);
   60: [XIC(Estop_Bulk) ,XIC(_JISdebug.0) XIC(Local:1:I.Data[48].21) ]OTE(DispersionAlarms[85]);
   61: [XIO(MCR_Bulk) ,XIC(_JISdebug.0) XIO(Local:1:I.Data[48].20) ]OTE(DispersionAlarms[86]);
   62: [XIC(LAH_S4352_1) ,XIC(_JISdebug.0) XIC(Local:1:I.Data[41].29) ]TON(D_AlarmTimers[87],?,?)XIC(D_AlarmTimers[87].DN)OTE(DispersionAlarms[87]);
   63: [XIC(LS_T53_High) ,XIC(_JISdebug.0) XIC(Local:1:I.Data[41].28) ]TON(D_AlarmTimers[88],?,?)XIC(D_AlarmTimers[88].DN)OTE(DispersionAlarms[88]);
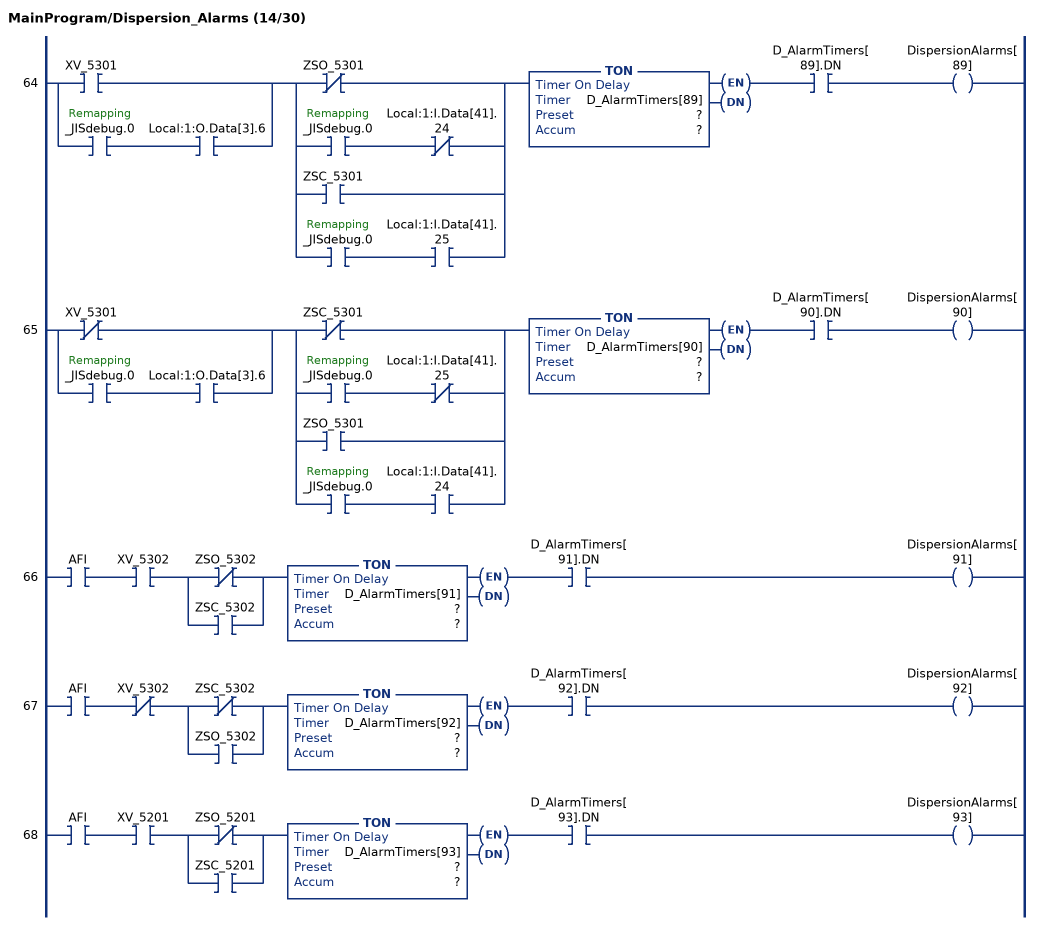
   64: [XIC(XV_5301) ,XIC(_JISdebug.0) XIC(Local:1:O.Data[3].6) ][XIO(ZSO_5301) ,XIC(_JISdebug.0) XIO(Local:1:I.Data[41].24) ,XIC(ZSC_5301) ,XIC(_JISdebug.0) XIC(Local:1:I.Data[41].25) ]TON(D_AlarmTimers[89],?,?)XIC(D_AlarmTimers[89].DN)OTE(DispersionAlarms[89]);
   65: [XIO(XV_5301) ,XIC(_JISdebug.0) XIC(Local:1:O.Data[3].6) ][XIO(ZSC_5301) ,XIC(_JISdebug.0) XIO(Local:1:I.Data[41].25) ,XIC(ZSO_5301) ,XIC(_JISdebug.0) XIC(Local:1:I.Data[41].24) ]TON(D_AlarmTimers[90],?,?)XIC(D_AlarmTimers[90].DN)OTE(DispersionAlarms[90]);
   66: XIC(AFI)XIC(XV_5302)[XIO(ZSO_5302) ,XIC(ZSC_5302) ]TON(D_AlarmTimers[91],?,?)XIC(D_AlarmTimers[91].DN)OTE(DispersionAlarms[91]);
   67: XIC(AFI)XIO(XV_5302)[XIO(ZSC_5302) ,XIC(ZSO_5302) ]TON(D_AlarmTimers[92],?,?)XIC(D_AlarmTimers[92].DN)OTE(DispersionAlarms[92]);
   68: XIC(AFI)XIC(XV_5201)[XIO(ZSO_5201) ,XIC(ZSC_5201) ]TON(D_AlarmTimers[93],?,?)XIC(D_AlarmTimers[93].DN)OTE(DispersionAlarms[93]);
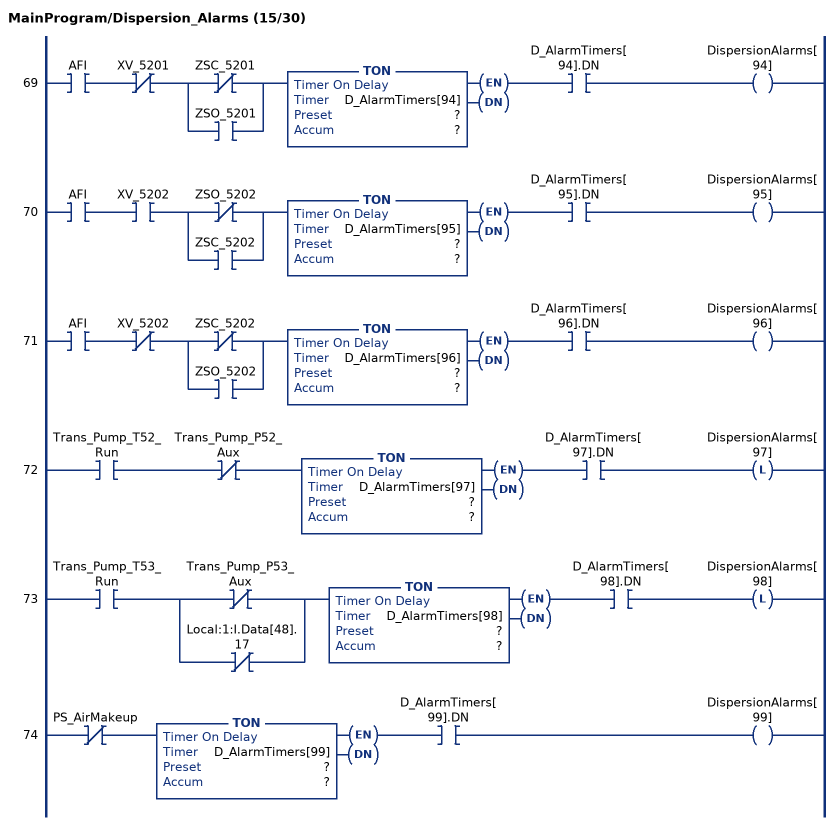
   69: XIC(AFI)XIO(XV_5201)[XIO(ZSC_5201) ,XIC(ZSO_5201) ]TON(D_AlarmTimers[94],?,?)XIC(D_AlarmTimers[94].DN)OTE(DispersionAlarms[94]);
   70: XIC(AFI)XIC(XV_5202)[XIO(ZSO_5202) ,XIC(ZSC_5202) ]TON(D_AlarmTimers[95],?,?)XIC(D_AlarmTimers[95].DN)OTE(DispersionAlarms[95]);
   71: XIC(AFI)XIO(XV_5202)[XIO(ZSC_5202) ,XIC(ZSO_5202) ]TON(D_AlarmTimers[96],?,?)XIC(D_AlarmTimers[96].DN)OTE(DispersionAlarms[96]);
   72: XIC(Trans_Pump_T52_Run)XIO(Trans_Pump_P52_Aux)TON(D_AlarmTimers[97],?,?)XIC(D_AlarmTimers[97].DN)OTL(DispersionAlarms[97]);
   73: XIC(Trans_Pump_T53_Run)[XIO(Trans_Pump_P53_Aux) ,XIO(Local:1:I.Data[48].17) ]TON(D_AlarmTimers[98],?,?)XIC(D_AlarmTimers[98].DN)OTL(DispersionAlarms[98]);
   74: XIO(PS_AirMakeup)TON(D_AlarmTimers[99],?,?)XIC(D_AlarmTimers[99].DN)OTE(DispersionAlarms[99]);
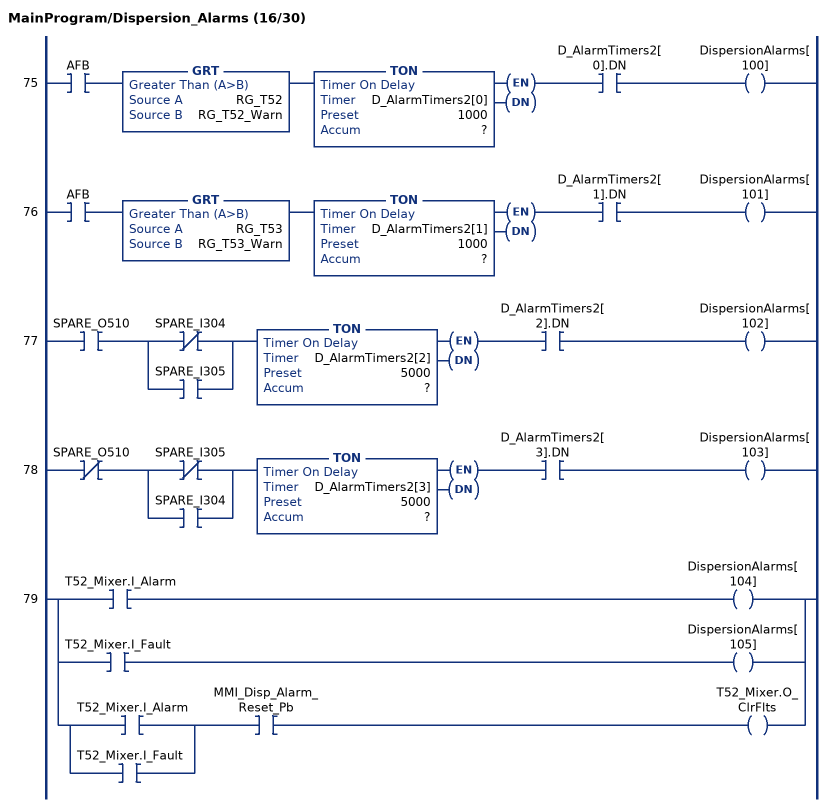
   75: XIC(AFB)GRT(RG_T52,RG_T52_Warn)TON(D_AlarmTimers2[0],?,?)XIC(D_AlarmTimers2[0].DN)OTE(DispersionAlarms[100]);
   76: XIC(AFB)GRT(RG_T53,RG_T53_Warn)TON(D_AlarmTimers2[1],?,?)XIC(D_AlarmTimers2[1].DN)OTE(DispersionAlarms[101]);
   77: XIC(SPARE_O510)[XIO(SPARE_I304) ,XIC(SPARE_I305) ]TON(D_AlarmTimers2[2],?,?)XIC(D_AlarmTimers2[2].DN)OTE(DispersionAlarms[102]);
   78: XIO(SPARE_O510)[XIO(SPARE_I305) ,XIC(SPARE_I304) ]TON(D_AlarmTimers2[3],?,?)XIC(D_AlarmTimers2[3].DN)OTE(DispersionAlarms[103]);
   79: [XIC(T52_Mixer.I_Alarm) OTE(DispersionAlarms[104]) ,XIC(T52_Mixer.I_Fault) OTE(DispersionAlarms[105]) ,[XIC(T52_Mixer.I_Alarm) ,XIC(T52_Mixer.I_Fault) ] XIC(MMI_Disp_Alarm_Reset_Pb) OTE(T52_Mixer.O_ClrFlts) ];
